# EPICS substitutions: iocBoot/ioc-tst-gige3/ioc-tst-gige3.substitutions
#
# GigE IOC archive substitutions file
#

# Generate IOC archive request
file archive_gige.archive
{
    {
        IOC = TST:R40:IOC:18,
    }
}
